// 
// 
// GVL_Persistent.stStatistics.udiTotalCycles :=
//     GVL_Persistent.stStatistics.aNest[1].udiTotalTests
//     + GVL_Persistent.stStatistics.aNest[2].udiTotalTests
//     + GVL_Persistent.stStatistics.aNest[3].udiTotalTests
//     + GVL_Persistent.stStatistics.aNest[4].udiTotalTests;
// 
// GVL_Persistent.stStatistics.udiTotalPass :=
//     GVL_Persistent.stStatistics.aNest[1].udiGoodParts
//     + GVL_Persistent.stStatistics.aNest[2].udiGoodParts
//     + GVL_Persistent.stStatistics.aNest[3].udiGoodParts
//     + GVL_Persistent.stStatistics.aNest[4].udiGoodParts;
// 
// GVL_Persistent.stStatistics.udiTotalFail :=
//     GVL_Persistent.stStatistics.aNest[1].udiBadParts
//     + GVL_Persistent.stStatistics.aNest[2].udiBadParts
//     + GVL_Persistent.stStatistics.aNest[3].udiBadParts
//     + GVL_Persistent.stStatistics.aNest[4].udiBadParts;
// 	
	
	
// =========================================================
// ACTIVE FAULT SUMMARY FOR MAIN HMI GRID
// =========================================================

// This summary represents only the faults currently responsible for the
// machine Fault state. The Events system keeps the complete alarm history
// independently for the dedicated Alarm page.
IF eMachineState = E_MachineState.Fault THEN

    stStatus.stAlarms.bHasFault := TRUE;
    stStatus.stAlarms.bHasSafetyStopFault := NOT stInputs.stSafety.bSafetyOk;

    stStatus.stAlarms.uiActiveCount := 0;

    IF NOT stInputs.stSafety.bSafetyOk THEN
        stStatus.stAlarms.uiActiveCount := stStatus.stAlarms.uiActiveCount + 1;
    END_IF

    IF bInitialisationTimeoutFault THEN
        stStatus.stAlarms.uiActiveCount := stStatus.stAlarms.uiActiveCount + 1;
    END_IF

    IF bStoppingTimeoutFault THEN
        stStatus.stAlarms.uiActiveCount := stStatus.stAlarms.uiActiveCount + 1;
    END_IF
	IF fbSiliconeSupportCylinder.IsFaulted() THEN
		stStatus.stAlarms.uiActiveCount := stStatus.stAlarms.uiActiveCount + 1;
	END_IF
	
	IF fbAssemblySupportCylinder.IsFaulted() THEN
		stStatus.stAlarms.uiActiveCount := stStatus.stAlarms.uiActiveCount + 1;
	END_IF

    IF fbAssemblyStation.IsFaulted() THEN
        stStatus.stAlarms.uiActiveCount := stStatus.stAlarms.uiActiveCount + 1;
    END_IF
    IF fbMainDoorLock.IsFaulted() THEN
        stStatus.stAlarms.uiActiveCount := stStatus.stAlarms.uiActiveCount + 1;
    END_IF

    IF fbIndex.IsFaulted() THEN
        stStatus.stAlarms.uiActiveCount := stStatus.stAlarms.uiActiveCount + 1;
    END_IF

    IF fbProcessStation.IsFaulted() THEN
        stStatus.stAlarms.uiActiveCount := stStatus.stAlarms.uiActiveCount + 1;
    END_IF

    IF ipEquipment.IsFaulted() THEN
        stStatus.stAlarms.uiActiveCount := stStatus.stAlarms.uiActiveCount + 1;
    END_IF

    IF stInputs.bEventFault THEN
        stStatus.stAlarms.uiActiveCount := stStatus.stAlarms.uiActiveCount + 1;
    END_IF

ELSE

    // Clear only the active-fault summary used by the main screen.
    // Do not acknowledge, clear or delete the Events history here.
    stStatus.stAlarms.bHasFault := FALSE;
    stStatus.stAlarms.bHasSafetyStopFault := FALSE;
    stStatus.stAlarms.uiActiveCount := 0;

END_IF

stStatus.stAlarms.eHighestAlarm 			:= E_AlarmId.None;
stStatus.aNest 								:= fbNestManager.GetAllNests();
stStatus.aNestStatistics 					:= fbNestManager.GetAllNestStatistics();
stStatus.udiAlarmCode 						:= 0;
stStatus.sOperatorMessage 					:= fbOperatorStation.GetMessage();

// =========================================================
// MACHINE MESSAGE SELECTION
// =========================================================

// Row 0 of the event DataGrid is exclusively the current automatic-cycle instruction.
IF eMachineState = E_MachineState.AutoCycle THEN

    IF stIndexStatus.eState = E_IndexState.WrongPositionRecovery THEN
        stStatus.sMachineMessage :='Index wrong position - place both hands on the safety controls to recover';

    ELSIF stProcessCycleStatus.eState = E_CycleState.WaitingForProcessesComplete THEN
		 stStatus.sMachineMessage :=stProcessCycleStatus.sMessage;
		 
    ELSIF fbOperatorStation.GetInstruction() <> E_OperatorInstruction.None THEN
        stStatus.sMachineMessage :=fbOperatorStation.GetMessage();
		
    ELSE
        stStatus.sMachineMessage := stProcessCycleStatus.sMessage;

    END_IF
	
ELSIF eMachineState = E_MachineState.Manual THEN
    stStatus.sMachineMessage := stManualModeStatus.sMessage;
	
ELSIF eMachineState = E_MachineState.Initialising THEN
    CASE eInitialisingWaitReason OF
		E_InitialisingWaitReason.MainDoorNotReady:stStatus.sMachineMessage 			:='System initialising - waiting for main door to lock';
        E_InitialisingWaitReason.SafetyNotReady: stStatus.sMachineMessage			:= 'System initialising - waiting for Safety OK';
        E_InitialisingWaitReason.FsoeNotReady: stStatus.sMachineMessage 			:= 'System initialising - waiting for FSoE';
        E_InitialisingWaitReason.SafetyLogicNotReady: stStatus.sMachineMessage 		:= 'System initialising - waiting for TwinSAFE logic';
        E_InitialisingWaitReason.IndexBusy: stStatus.sMachineMessage 				:= 'System initialising - waiting for index to stop';
        E_InitialisingWaitReason.SiliconeSupportNotRetracted:stStatus.sMachineMessage := 'System initialising - waiting for Silicone Support Cylinder retract';
		E_InitialisingWaitReason.AssemblySupportNotRetracted:stStatus.sMachineMessage := 'System initialising - waiting for Assembly Support Cylinder retract';
		E_InitialisingWaitReason.SiliconeSupportFaulted:stStatus.sMachineMessage 	:= 'System initialising - Silicone Support Cylinder fault';
		E_InitialisingWaitReason.AssemblySupportFaulted: stStatus.sMachineMessage 	:= 'System initialising - Assembly Support Cylinder fault';
        E_InitialisingWaitReason.AssemblyStationNotHome: stStatus.sMachineMessage   := stAssemblyStationStatus.sMessage;
        E_InitialisingWaitReason.AssemblyStationFaulted: stStatus.sMachineMessage   := 'System initialising - assembly station fault';
        E_InitialisingWaitReason.ProcessStationFaulted: stStatus.sMachineMessage 	:= 'System initialising - process station fault';
        E_InitialisingWaitReason.MainDoorFaulted: stStatus.sMachineMessage 			:= 'System initialising - main door lock fault';
        E_InitialisingWaitReason.ProcessEquipmentNotReady: stStatus.sMachineMessage := 'System initialising - waiting for process equipment';
   		E_InitialisingWaitReason.AirSupplyNotReady:stStatus.sMachineMessage 		:= 'System initialising - waiting for air supply';
		E_InitialisingWaitReason.ExtractorNotReady:stStatus.sMachineMessage 		:= 'System initialising - waiting for vacuum extractor';


 ELSE stStatus.sMachineMessage 													:= 'System initialising'; 
		
		
		
END_CASE
	
ELSIF eMachineState = E_MachineState.ReadyToStart THEN

    IF stInputs.eIndexPosition = E_TablePosition.Unknown THEN
        stStatus.sMachineMessage :='Index wrong position - press Start to recover in Auto Cycle';

    ELSE
        stStatus.sMachineMessage :='Ready to start';

    END_IF
	
	
ELSIF eMachineState = E_MachineState.Stopping THEN
    CASE eStoppingWaitReason OF
        E_StoppingWaitReason.IndexStillMoving:stStatus.sMachineMessage := 'System stopping - waiting for index';
        E_StoppingWaitReason.SiliconeSupportRetracting:stStatus.sMachineMessage := 'System stopping - retracting Silicone Support Cylinder';
		E_StoppingWaitReason.AssemblySupportRetracting: stStatus.sMachineMessage := 'System stopping - retracting Assembly Support Cylinder';
        E_StoppingWaitReason.ProcessEquipmentStopping:stStatus.sMachineMessage := 'System stopping - stopping process equipment';
        E_StoppingWaitReason.MainDoorTransition:stStatus.sMachineMessage := 'System stopping - waiting for main door transition';
    ELSE
        stStatus.sMachineMessage := 'System stopping';
    END_CASE
	
	
ELSIF eMachineState = E_MachineState.Fault THEN

    IF NOT stInputs.stSafety.bSafetyOk THEN

        stStatus.sMachineMessage :='Machine fault - safety system not ready';

    // ---------------------------------------------------------
    // SILICONE SUPPORT FAULT
    // ---------------------------------------------------------

    ELSIF fbSiliconeSupportCylinder.IsFaulted() THEN

        stStatus.sMachineMessage :='Machine fault - Silicone Support Cylinder feedback fault';


    // ---------------------------------------------------------
    // ASSEMBLY SUPPORT FAULT
    // ---------------------------------------------------------

    ELSIF fbAssemblySupportCylinder.IsFaulted() THEN

        stStatus.sMachineMessage := 'Machine fault - Assembly Support Cylinder feedback fault';


    // ---------------------------------------------------------
    // ASSEMBLY / FLIPPING STATION FAULT
    // ---------------------------------------------------------

    ELSIF fbAssemblyStation.IsFaulted() THEN

        stStatus.sMachineMessage :='Machine fault - assembly/flipping station fault';


    // ---------------------------------------------------------
    // INITIALISATION TIMEOUT
    // ---------------------------------------------------------

    ELSIF bInitialisationTimeoutFault THEN

        CASE eInitialisingWaitReason OF

            E_InitialisingWaitReason.AirSupplyNotReady:stStatus.sMachineMessage := 'Initialisation timeout - air supply not ready';
			E_InitialisingWaitReason.ExtractorNotReady:stStatus.sMachineMessage :='Initialisation timeout - vacuum extractor not running';
            E_InitialisingWaitReason.IndexBusy:stStatus.sMachineMessage := 'Initialisation timeout - index did not stop';
            E_InitialisingWaitReason.SiliconeSupportNotRetracted:stStatus.sMachineMessage := 'Initialisation timeout - Silicone Support Cylinder not retracted';
            E_InitialisingWaitReason.AssemblySupportNotRetracted: stStatus.sMachineMessage := 'Initialisation timeout - Assembly Support Cylinder not retracted';
            E_InitialisingWaitReason.SiliconeSupportFaulted:stStatus.sMachineMessage := 'Initialisation timeout - Silicone Support Cylinder fault';
            E_InitialisingWaitReason.AssemblySupportFaulted:stStatus.sMachineMessage := 'Initialisation timeout - Assembly Support Cylinder fault';
            E_InitialisingWaitReason.AssemblyStationNotHome:stStatus.sMachineMessage := 'Initialisation timeout - assembly station did not reach home position';
            E_InitialisingWaitReason.AssemblyStationFaulted:stStatus.sMachineMessage := 'Initialisation timeout - assembly station fault';
            E_InitialisingWaitReason.MainDoorFaulted:stStatus.sMachineMessage := 'Initialisation timeout - main door lock fault';
            E_InitialisingWaitReason.MainDoorNotReady: stStatus.sMachineMessage := 'Initialisation timeout - main door did not lock';
            E_InitialisingWaitReason.ProcessStationFaulted:stStatus.sMachineMessage := 'Initialisation timeout - process station fault';
            E_InitialisingWaitReason.ProcessEquipmentNotReady:stStatus.sMachineMessage := 'Initialisation timeout - process equipment not ready';
			E_InitialisingWaitReason.IvekHeaterNotReady:stStatus.sMachineMessage :='System initialising - IVEK heater controller alarm';
      
		ELSE

            stStatus.sMachineMessage := 'Machine fault - initialisation timeout';

        END_CASE
    ELSIF bStoppingTimeoutFault THEN
        CASE eStoppingWaitReason OF
            E_StoppingWaitReason.IndexStillMoving:
                stStatus.sMachineMessage := 'Stopping timeout - index still moving';
            E_StoppingWaitReason.SiliconeSupportRetracting:
                stStatus.sMachineMessage := 'Stopping timeout - Silicone Support Cylinder not retracted';
			E_StoppingWaitReason.AssemblySupportRetracting:
                stStatus.sMachineMessage := 'Stopping timeout - Assembly Support Cylinder not retracted';
            E_StoppingWaitReason.ProcessEquipmentStopping:
                stStatus.sMachineMessage := 'Stopping timeout - process equipment still running';
            E_StoppingWaitReason.MainDoorTransition:
                stStatus.sMachineMessage := 'Stopping timeout - main door transition incomplete';
        ELSE
            stStatus.sMachineMessage := 'Machine fault - stopping timeout';
        END_CASE
		
	ELSIF stProcessCycleStatus.bFaulted THEN
   	 	stStatus.sMachineMessage := stProcessCycleStatus.sMessage;
    ELSIF fbMainDoorLock.IsFaulted() THEN
        stStatus.sMachineMessage := 'Machine fault - main door lock fault';
    ELSIF fbIndex.IsFaulted() THEN
        stStatus.sMachineMessage := 'Machine fault - index table fault';
    ELSIF fbProcessStation.IsFaulted() THEN
        stStatus.sMachineMessage := 'Machine fault - process station fault';
    ELSIF ipEquipment.IsFaulted() THEN
        stStatus.sMachineMessage := 'Machine fault - process equipment fault';
    ELSIF stInputs.bEventFault THEN
        stStatus.sMachineMessage := 'Machine fault - check active alarms';
    ELSE
        stStatus.sMachineMessage := 'Machine fault - reset required';
    END_IF
ELSIF eMachineState = E_MachineState.Stopped THEN
    IF GVL_HMI.bIvekSettingsInterlock THEN
        stStatus.sMachineMessage := 'Machine stopped - IVEK configuration interface active';

    ELSIF NOT stSiliconeSupplyStatus.bSelectedReservoirReady THEN
        stStatus.sMachineMessage := 'Silicone supply not ready - configure reservoir in Settings';

    ELSIF NOT stInputs.bMainDoorClosed THEN
        stStatus.sMachineMessage := 'Machine stopped - close the main door and press Reset';

    ELSE
        stStatus.sMachineMessage := 'Machine stopped - press Reset to initialise';
    END_IF
ELSE
    stStatus.sMachineMessage := 'Machine stopped';
END_IF

// =========================================================
// END-OF-CYCLE STATE AND OUTPUT PUBLICATION
// =========================================================

IF eMachineState <> E_MachineState.Manual
AND NOT fbSiliconeProcess.IsBusy() THEN
    bManualSiliconeCycleActive := FALSE;
END_IF

IF eMachineState <> E_MachineState.Manual
AND NOT fbAssemblyStation.IsBusy() THEN
    bManualAssemblyCycleActive := FALSE;
END_IF

//ePreviousMachineState := eMachineState;
stOutputs := stOutputsInternal;
END_METHOD

METHOD PRIVATE ResetCyclicOutputs
stOutputsInternal.bSafetyRunRequest := FALSE;
stOutputsInternal.bSafetyResetRequest := FALSE;
stOutputsInternal.bAirSupplyEnable := FALSE;
stOutputsInternal.bIndexRotatePortA := FALSE;
stOutputsInternal.bIndexStopPortB := FALSE;
stOutputsInternal.bAssemblySupportExtend := FALSE;
stOutputsInternal.bAssemblySupportRetract := TRUE;
stOutputsInternal.bSiliconeSupportExtend := FALSE;
stOutputsInternal.bSiliconeSupportRetract := TRUE;
stOutputsInternal.bTransferVerticalMiniSlideExtend := FALSE;
stOutputsInternal.bTransferVerticalMiniSlideRetract := FALSE;
stOutputsInternal.bRotaryGripperOpen := FALSE;
stOutputsInternal.bRotaryGripperClose := FALSE;
stOutputsInternal.bRotaryGripperRotationPick0 := FALSE;
stOutputsInternal.bRotaryGripperRotationPlace180 := FALSE;
stOutputsInternal.bMainDoorLockRequest := FALSE;
stOutputsInternal.bLedStart := FALSE;
stOutputsInternal.bLedReset := FALSE;
stOutputsInternal.bLedPass := FALSE;
stOutputsInternal.bLedFail := FALSE;
stOutputsInternal.bInternalLight := FALSE;
stOutputsInternal.bPuckLockerPinUp := FALSE;
stOutputsInternal.bSiliconeAirEnable := FALSE;
END_METHOD

END_FUNCTION_BLOCK

(* stored: Version 1.1.0.1, ProductVersion 3.1.4026.18
   POU FB_IndexedSiliconeMachine: Id {ff07b0ce-3073-475d-ae18-b3b039ab22f1}, SpecialFunc None
   Method CheckComponentFaults: Id {1e0a6e8d-fb2f-4560-a186-ac64f265cfd0}
   Method Cyclic: Id {b3ad9d70-3bf2-42da-ab5a-7255e3c227a5}
   Method ResetCyclicOutputs: Id {9b31b272-cf95-4c0b-9674-4eee2c2eaa71} *)
